// TwinCAT 3 PLC project lcls_twincat_motion_unit_tests_PLC
// ProgramVersion: 3.1.4022.3
// libraries:
//   lcls-twincat-motion-gantry-lib-sheppard, * (SLAC)
//   Tc2_MC2, * (Beckhoff Automation GmbH)
//   Tc2_Standard, * (Beckhoff Automation GmbH)
//   Tc2_System, * (Beckhoff Automation GmbH)
//   Tc3_Module, * (Beckhoff Automation GmbH)
//   TcUnit,0.0.0.0,www.tcunit.org
// project tree:
//   GVLs/ TestAxes.TcGVL
//   / PlcTask.TcTTO
//   POUs/ MAIN.TcPOU
//   POUs/Test/ FB_GantryAutoCoupling_Test.TcPOU, PRG_TEST.TcPOU
// real-time tasks:
//   TASK PlcTask: cycle T#10ms, priority 20, ADS port 350
// motion (NC):
//   TASK NC-Task 1 SAF: cycle T#2ms, priority 4, ADS port 501
//   TASK NC-Task 1 SVB: cycle T#10ms, priority 8, ADS port 511
//   AXIS Axis_M1 (id 1)
//   AXIS Axis_M2 (id 2)
// variable links:
//   lcls_twincat_motion_unit_tests_PLC Instance <-> NC-Task 1 SAF/Axes/Axis_M1
//     PlcTask Inputs/TestAxes.M1.Axis.NcToPlc <-> Outputs/ToPlc
//     PlcTask Outputs/TestAxes.M1.Axis.PlcToNc <-> Inputs/FromPlc
//   lcls_twincat_motion_unit_tests_PLC Instance <-> NC-Task 1 SAF/Axes/Axis_M2
//     PlcTask Inputs/TestAxes.M2.Axis.NcToPlc <-> Outputs/ToPlc
//     PlcTask Outputs/TestAxes.M2.Axis.PlcToNc <-> Inputs/FromPlc

CONFIGURATION lcls_twincat_motion_unit_tests_PLC
    RESOURCE PLC ON TwinCAT3
        TASK PlcTask(INTERVAL := T#10ms, PRIORITY := 20);
        PROGRAM PRG_TEST WITH PlcTask : PRG_TEST;
    END_RESOURCE
END_CONFIGURATION

// ---- GVLs/TestAxes.TcGVL
{attribute 'qualified_only'}
VAR_GLOBAL
	M1 : DUT_MotionStage:=(nEnableMode:=0); // Test Master Axis
	master_enc : ST_RenishawAbsEnc;

	M2 : DUT_MotionStage:=(nEnableMode:=0); // Test Slave Axis
	slave_enc : ST_RenishawAbsEnc;
END_VAR

// ---- POUs/Test/PRG_TEST.TcPOU
PROGRAM PRG_TEST
VAR
	fbGantryAutoCoupling_Test : FB_GantryAutoCoupling_Test;
END_VAR

TcUnit.RUN();

END_PROGRAM

// ---- POUs/Test/FB_GantryAutoCoupling_Test.TcPOU
{attribute 'call_after_init'}
FUNCTION_BLOCK FB_GantryAutoCoupling_Test EXTENDS TcUnit.FB_TestSuite

CoupledOnStartup();

METHOD PRIVATE CoupledOnStartup
VAR_INST
	fbAutoCouple : FB_GantryAutoCoupling;

	// @TEST-FIXTURE EmergencyErrorCode
	fbMotionStage_M1, fbMotionStage_M2 : FB_MotionStage;

	nCycleCount : ULINT := 0;
END_VAR
VAR
	bStartCouple : BOOL;
	bStopCouple : BOOL;

	// @TEST-RESULT CouplingStatus
	ExpectedStatus : BOOL := TRUE;
	WatchCouplingStatus : BOOL;
	CouplingStatus : BOOL;
END_VAR
TEST('CoupledOnStartup');

nCycleCount := nCycleCount + 1;

TestAxes.M1.bGantryAxis := TRUE;
TestAxes.M1.fGantryTol := 50000;
TestAxes.M1.nCommand := 3;
TestAxes.M2.bGantryAxis := TRUE;
TestAxes.M2.fGantryTol := TestAxes.M1.fGantryTol;

TestAxes.master_enc.Count := LREAL_TO_ULINT(TestAxes.M1.stAxisStatus.fActPosition * EXPT(10, 6));
TestAxes.slave_enc.Count := LREAL_TO_ULINT(TestAxes.M1.stAxisStatus.fActPosition * EXPT(10, 6));

// @TEST-RUN
fbMotionStage_M1(stMotionStage:=TestAxes.M1);
fbMotionStage_M2(stMotionStage:=TestAxes.M2);

WatchCouplingStatus := TestAxes.M1.Axis.NcToPlc.CoupleState=1 AND TestAxes.M2.Axis.NcToPlc.CoupleState=3;



fbAutoCouple(fGantryTol:=5000, Master:=TestAxes.M1, MasterEnc:=TestAxes.master_enc, Slave:=TestAxes.M2,
	         SlaveEnc:=TestAxes.slave_enc, bExecuteCouple:=bStartCouple,
			 bExecuteDecouple:=bStopCouple,
			 bGantryAlreadyCoupled=>CouplingStatus);

IF nCycleCount = 2 THEN
	// @TEST-ASSERT
	AssertEquals(Expected:=ExpectedStatus, Actual:=CouplingStatus,
	         	 Message:='Master and Slave did not start coupled');

	TEST_FINISHED('');
END_IF
END_METHOD

END_FUNCTION_BLOCK

// ---- POUs/MAIN.TcPOU
PROGRAM MAIN
VAR
END_VAR

END_PROGRAM
